INTERFACE IVisitorHandler

METHOD subscribe : BOOL
VAR_INPUT
	subscriber: IVisitor;
END_VAR
END_METHOD

METHOD unSubscribe : BOOL
VAR_INPUT
	subscriber: IVisitor;
END_VAR
END_METHOD

END_INTERFACE

(* stored: Version 1.1.0.1
   Itf IVisitorHandler: Id {27e35cdd-c5bf-4c2a-b6d0-6293849fbcc8}
   Method subscribe: Id {281fe6a7-c3c0-4b3a-b839-73f4c35fd384}
   Method unSubscribe: Id {b5d76387-ffa7-42fd-af93-cc339f812700} *)
